// Mitsubishi GX Works2 project: q01   PLC: Q02/Q02H

PROGRAM MAIN
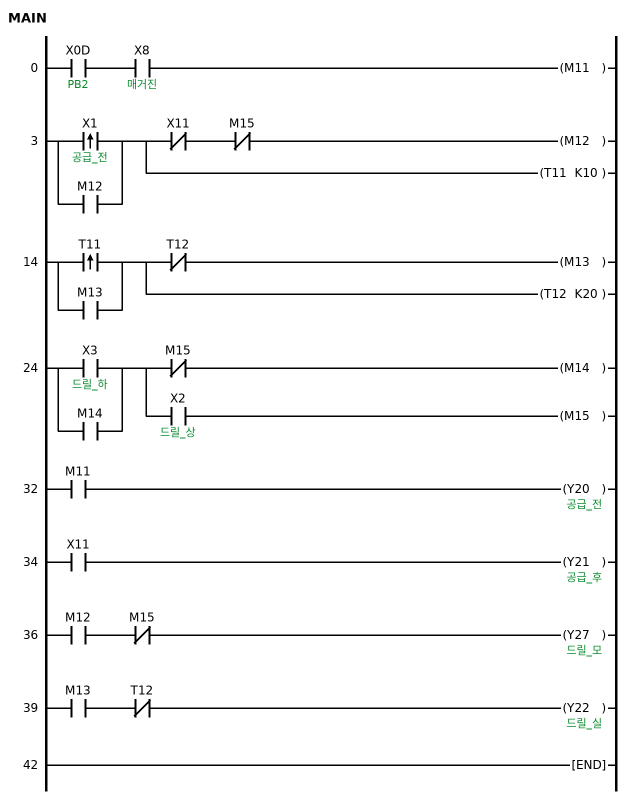
0     LD      X0D  ; PB2
      AND     X8  ; 매거진
      OUT     M11
3     LDP     X1  ; 공급_전
      OR      M12
      MPS
      ANI     X11
      ANI     M15
      OUT     M12
      MPP
      OUT     T11 K10
14    LDP     T11
      OR      M13
      MPS
      ANI     T12
      OUT     M13
      MPP
      OUT     T12 K20
24    LD      X3  ; 드릴_하
      OR      M14
      MPS
      ANI     M15
      OUT     M14
      MPP
      AND     X2  ; 드릴_상
      OUT     M15
32    LD      M11
      OUT     Y20  ; 공급_전
34    LD      X11
      OUT     Y21  ; 공급_후
36    LD      M12
      ANI     M15
      OUT     Y27  ; 드릴_모
39    LD      M13
      ANI     T12
      OUT     Y22  ; 드릴_실
42    END
END_PROGRAM

// device comments not shown above
X0  ; 공급_후
X4  ; 송출_후
X5  ; 송출_전
X6  ; 배출_후
X7  ; 배출_전
X9  ; 이송감지
X0A  ; 비금속
X0B  ; 금속
X0C  ; PB1
X0E  ; PB3
X0F  ; 비상정지
Y23  ; 송출_전
Y24  ; 송출_후
Y25  ; 배출_전
Y26  ; 배출_후
Y28  ; 컨베
Y29  ; 적램
Y2A  ; 황램
Y2B  ; 녹램
